(* CoDeSys 2.3 export: CLOCKPULSES.EXP *)

(* Global variable list: ClockPulses *)
VAR_GLOBAL
	_CLOCK_100MS AT %QX0.0: BOOL ;
	_CLOCK_1S AT %QX0.1: BOOL ;
	_CLOCK_10S AT %QX0.2: BOOL ;
	_CLOCK_60S AT %QX0.3: BOOL ;
END_VAR
